FUNCTION_BLOCK fbInheritanceLevel_3 EXTENDS fbInheritanceLevel_2
VAR
	{attribute addProperty Name "LEVEL 3"}
	level_3 : stAllTypes;
END_VAR

SUPER^();

METHOD Init : BOOL
VAR_INPUT
END_VAR
SUPER^.Init();
END_METHOD

END_FUNCTION_BLOCK

(* stored: Version 1.1.0.1, ProductVersion 3.1.4022.7
   POU fbInheritanceLevel_3: Id {0cf8711d-2409-47a3-aeff-3b639be91487}, SpecialFunc None
   Method Init: Id {48c2de65-8514-428f-8818-6a0d3d15dff1} *)
